TYPE ST_BeamParams :
STRUCT
	// Beam parameters
	// These must be filled in by the caller.
	
	//Note: fAtt is a local parameter, meaning it is distributed to the nearest
	// upstream attenuator component.
	fAtt : REAL := 100; //Requested attenuation %
	
	//Machine parameters
	nRate	:	UINT	:= 10; //Pulse-rate
	fPP_mJ : REAL := 20; //Requested per pulse max energy (mJ)
	fUpper_eV	:	REAL	:= 20000; //Requested max eV
	fLower_eV	:	REAL	:= 0; //Requested lower eV
END_STRUCT
END_TYPE

(* stored: Version 1.1.0.1, ProductVersion 3.1.4022.12
   DUT ST_BeamParams: Id {1cfc4571-cdd9-4483-b0d1-cbcb7d03cd4c} *)
